# EPICS autosave request: profile_bluesky/startup/ref/Db/stringout_settings.req
# FILE... stringout_settings.req
# USAGE... stringout Record fields autosave'd.
$(P).DESC
$(P).VAL
